// TIA Portal project "time_error_interrupt" (V18)

(* hardware
DEVICE "S7-1200 station_1"  S7-1200 Station
   slot 0: "Rack_0"  S7-1200 Rack  Rack  V1.0
   slot 1: "PLC_1"  CPU 1214C DC/DC/DC  6ES7 214-1AG40-0XB0  V4.6
*)

// ===== PLC "PLC_1"  CPU 1214C DC/DC/DC =====

VAR_GLOBAL   // PLC tag table "Default tag table"
   "Tag_1" AT %I0.0 : Bool;
   "Tag_2" AT %M100.0 : Bool;
   "Tag_3" AT %MD0 : DWord;
END_VAR

ORGANIZATION_BLOCK "Main"   // OB1, LAD, ProgramCycle
TITLE = "Main Program Sweep (Cycle)"
{ S7_Optimized_Access := 'TRUE' }
VERSION : 0.1
   VAR_INPUT
      Initial_Call : Bool;   // Initial call of this OB
      Remanence : Bool;   // =True, if remanent data are available
   END_VAR
   VAR_TEMP   // added for the SCL form of the ladder/FBD networks
      _w1 : Bool;
   END_VAR
BEGIN

REGION Network 1
   // positif kenar darbesi uygulanmalı
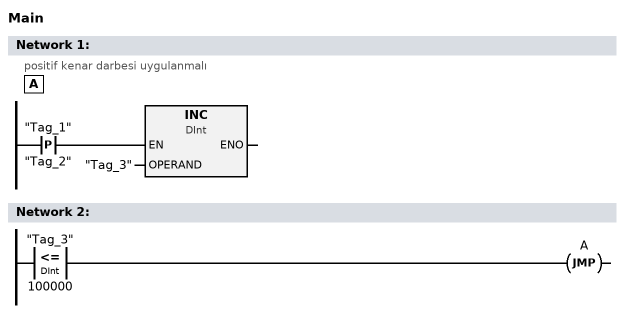
   Label( A )
   RUNG wire#powerrail
      P_Contact(operand := "Tag_1", bit := "Tag_2")
      { S7_Templates := "DestType := DInt" } Inc( "Tag_3" )
   END_RUNG
   // the same network as SCL:
   A:
   #_w1 := "Tag_1" AND NOT "Tag_2";   // rising edge of "Tag_1"
   "Tag_2" := "Tag_1";
   IF #_w1 THEN "Tag_3" := "Tag_3" + 1; END_IF;
END_REGION

REGION Network 2
   RUNG wire#powerrail
      { S7_Templates := "SrcType := DInt" } LE_Contact(in1 := "Tag_3", in2 := 100000)
      JumpCoil( A )
   END_RUNG
   // the same network as SCL:
   IF "Tag_3" <= 100000 THEN GOTO A; END_IF;
END_REGION
END_ORGANIZATION_BLOCK